{attribute 'qualified_only'}
TYPE E_AlarmCategory :
(
Configuration:= 1, 
Safety := 65536000,
TrackClient := 131072000,
OPCcomm := 196608000,
JobData := 262144000,
ConfigurationData := 327680000,
//GeneralSpare := 393216000,
//GeneralSpare := 458752000,
//GeneralSpare := 524288000,
//GeneralSpare := 589824000,
//GeneralSpare := 655360000,
OP11200 := 734003200,
OP11210 := 734658560,
OP11400 := 747110400,
OP11600 := 760217600,
OP11601 := 760283136,
OP11602 := 760348672,
OP11603 := 760414208,
OP11604 := 760479744,
OP11700 := 766771200,
OP12000 := 786432000,
OP12001 := 786497536,
OP12002 := 786563072,
OP12003 := 786628608,
OP12004 := 786694144,
OP12010 := 787087360,
OP12011 := 787152896,
OP12200 := 799539200,
OP12500 := 819200000,
OP12600 := 825753600,
OP12900 := 845414400,
OP12901 := 845479936,
OP12902 := 845545472,
OP12903 := 845611008,
OP12904 := 845676544,
OP12910 := 846069760,
OP12911 := 846135296,
OP12912 := 846200832,
OP12913 := 846266368,
OP12914 := 846331904,
OP13100 := 858521600,
OP13200 := 865075200,
OP13300 := 871628800,
OP13500 := 884736000,
OP13800 := 904396800,
OP16000 := 1048576000,
OP16100 := 1055129600,
OP16200 := 1061683200,
OP16300 := 1068236800,
OP16400 := 1074790400,
OP21900 := 1435238400,
OPSpare := 3276800000,
Robot := 3342336000,
LifterStation1Device := 3407872000,
LifterStation2Device := 3473408000,
LastingDevice := 3538944000
)UDINT;
END_TYPE

(* stored: Version 1.1.0.1, ProductVersion 3.1.4024.5
   DUT E_AlarmCategory: Id {5ea03c69-45e5-4b63-92c4-4b88f60de61c} *)
